// TIA Portal V20 export
TYPE "typeEmHomedCheck"
// stored: Access Published, Namespace Unit1.Em7
   STRUCT
      cmNgKickerAxisZ : Bool;
      cmPassKickerAxisZ : Bool;
      cmCutConveyorAxisB : Bool;
      cmNgConveyorAxisB : Bool;
      cmStack1ConveyorAxisB : Bool;
      cmStack2ConveyorAxisB : Bool;
      cmCutConveyorRingBlow : Bool;
      cmNgConveyorRingBlow : Bool;
      cmStack2ConveyorRingBlow : Bool;
      cmNgBoxLockCylinderUpDown : Bool;
      cmStack1QrReader : Bool;
      cmStack2QrReader : Bool;
   END_STRUCT;
END_TYPE
